FUNCTION_BLOCK VAV_MDLL (* Variable Air Valve Model with Local Comms *)
  (* Standard: 61499-1; Classification: Simulation; ApplicationDomain: HVAC; Function: Variable Air Valve *)
  (* Version 0.1, 2006-05-01, JHC, Holobloc Inc, Changed FV to FD. *)
  (* Version 0.0, 2006-04-12, JHC, Holobloc Inc *)
  (* Compiler header: package fb.rt.hvac; import fb.rt.net.*; import fb.rt.mva.*; *)
  (* Compiler classdef: public class VAV_MDLL extends FBMVCD *)
  (* Compiler Java Sun JDK 1.5.0 *)
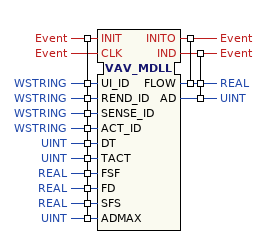
  EVENT_INPUT
    INIT WITH DT, TACT, FSF, FD, SFS, ADMAX, UI_ID, REND_ID, SENSE_ID, ACT_ID; (* Initialization *)
    CLK; (* VAV simulation clock *)
  END_EVENT
  EVENT_OUTPUT
    INITO WITH FLOW; (* Initialization complete *)
    IND WITH FLOW, AD; (* Follows every CLK event *)
  END_EVENT
  VAR_INPUT
    UI_ID : WSTRING; (* User input channel ID from View *)
    REND_ID : WSTRING; (* Rendering data channel ID to View *)
    SENSE_ID : WSTRING; (* Sensor data channel ID to Controller *)
    ACT_ID : WSTRING; (* Actuator Channel ID *)
    DT : UINT := 10; (* Clock period, sec *)
    TACT : UINT := 95; (* Damper actuation time, sec *)
    FSF : REAL := 1000.0; (* Air Flow at Damper Full Open, CFM *)
    FD : REAL; (* Maximum random flow deviation in CFM *)
    SFS : REAL := 1000.0; (* Air Flow at Sensor Full Scale, CFM *)
    ADMAX : UINT := 4096; (* Maximum Flow Sensor A/D converter value + 1, default is 12 bits *)
  END_VAR
  VAR_OUTPUT
    FLOW : REAL; (* Air flow, CFM *)
    AD : UINT; (* Flow sensor A/D converter value *)
  END_VAR
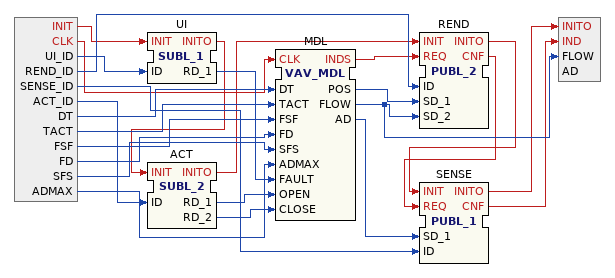
  FBS
    MDL : VAV_MDL;
    UI : SUBL_1;
    ACT : SUBL_2;
    REND : PUBL_2;
    SENSE : PUBL_1;
  END_FBS
  EVENT_CONNECTIONS
    UI.INITO TO ACT.INIT;
    ACT.INITO TO REND.INIT;
    MDL.INDS TO REND.REQ;
    REND.INITO TO SENSE.INIT;
    SENSE.INITO TO INITO;
    REND.CNF TO SENSE.REQ;
    SENSE.CNF TO IND;
    INIT TO UI.INIT;
    CLK TO MDL.CLK;
  END_CONNECTIONS
  DATA_CONNECTIONS
    DT TO MDL.DT;
    TACT TO MDL.TACT;
    FSF TO MDL.FSF;
    FD TO MDL.FD;
    SFS TO MDL.SFS;
    ADMAX TO MDL.ADMAX;
    UI.RD_1 TO MDL.FAULT;
    UI_ID TO UI.ID;
    ACT.RD_1 TO MDL.OPEN;
    ACT.RD_2 TO MDL.CLOSE;
    REND_ID TO REND.ID;
    MDL.POS TO REND.SD_1;
    MDL.FLOW TO REND.SD_2;
    MDL.FLOW TO FLOW;
    MDL.AD TO SENSE.SD_1;
    SENSE_ID TO SENSE.ID;
    ACT_ID TO ACT.ID;
  END_CONNECTIONS
END_FUNCTION_BLOCK
